# B&R Automation Studio project Stanze
Automation Studio 4.9

## Configuration Config1

CPU PC_any, AutomationRuntime C4.90, Build 4.1.2, Vc V4.72.2

### Task classes (Cpu.sw)
```
Cyclic#4:
  Program <- Program.prg
  Program1 <- Program1.prg
Libraries: standard
```

### Hardware
```
PC : PC_any v1.1.1.0 (OrderNumber=PC)
```

## Logical view

### Program Logical/Program (ANSIC)

#### Variables.var
```iecst
VAR
	T1 : TON;
	Richtung : BOOL;
	Motor : BOOL;
	Unten : BOOL;
	Start : BOOL;
	Schritt : USINT;
	Oben : USINT;
END_VAR
```

#### Main.c
```c
#include <bur/plctypes.h>

#ifdef _DEFAULT_INCLUDES
	#include <AsDefault.h>
#endif

void _INIT ProgramInit(void)
{
	T1.PT=3000;
}

void _CYCLIC ProgramCyclic(void)
{
	Motor=Richtung=0;

	switch(Schritt)
	{
		case 0:

			if(Start == 1)

			{ Schritt = 1; }

			break;

		case 1:

			Motor = 1;

			Richtung = 1;

			if(Unten == 1)

			{Schritt = 2;}

			break;

		case 2:

			T1.IN=1;
			if(T1.Q)

			{Schritt = 3;}

			break;

		case 3:

			Motor = 1;

			if(Oben == 1)

			{ Schritt = 0;}

			break;

	}

}

void _EXIT ProgramExit(void)
{

}
```

### Program Logical/Program1 (ANSIC)

#### Variables.var
```iecst
VAR
	Schritt : USINT;
	Ri : BOOL;
	S0 : BOOL;
	S1 : BOOL;
	S2 : BOOL;
	S3 : BOOL;
	V1 : BOOL;
	Y1 : BOOL;
	Y2 : BOOL;
	Q1 : BOOL;
	H1 : BOOL;
	T1 : TON;
END_VAR
```

#### Main.c
```c
#include <bur/plctypes.h>

#ifdef _DEFAULT_INCLUDES
	#include <AsDefault.h>
#endif

void _INIT ProgramInit(void)
{
	T1.PT=30000;
}

void _CYCLIC ProgramCyclic(void)
{
	TON(&T1); //Aufruf der Timerfunktion
	V1=Y1=Y2=H1=0;
	switch (Schritt) {
		case 0: if (S0)
			{
				Schritt=1;
			}
			break;
		case 1:
			V1=1;
			Y1=1;
			if (S2)
			{
				Schritt=2;
			}
			break;
		case 2:
			T1.IN=1;
			V1=1;
			if (S1&&T1.Q==0)
			{
				Schritt=4;
				T1.IN=0;
				T1.Q=0;
				T1.M=0;
			}
			else if (T1.Q)
			{
				Schritt=3;
				T1.IN=0;
				T1.Q=0;
				T1.M=0;
			}
			break;
		case 3:
			V1=1;
			Y2=1;
			if (S3)
			{
				Schritt=0;
			}
			break;
		case 4:
			H1=1;
			V1=1;
			Y2=1;
			if (S3)
			{
				Schritt=5;
			}
			break;
		case 5:
			H1=1;
			if (Q1)
			{
				Schritt=0;
			}
			break;
	}
}
void _EXIT ProgramExit(void)
{

}
```

Listed in the project but not available here: Logical/Global.typ, Logical/Global.var, Logical/Libraries
